PROGRAM PRG_MAIN
VAR
END_VAR

// NETWORK 1

END_PROGRAM

(* stored: Version 1.1.0.1
   POU PRG_MAIN: Id {3f14fd95-3576-417d-8629-e7ee356023c5}, SpecialFunc None *)
